(* IEC 61131-3 sources: Lasal/CPU_5344_V01/Class/Lees10Ingangenin, 1 file *)

(* ---- Lees10Ingangenin.st ---- *)
(*!
<Class
	Name               = "Lees10Ingangenin"
	Revision           = "0.0"
	RealtimeTask       = "false"
	CyclicTask         = "false"
	BackgroundTask     = "false"
	Sigmatek           = "false"
	OSInterface        = "false"
	HighPriority       = "false"
	Automatic          = "false"
	UpdateMode         = "Prescan"
	SharedCommandTable = "true"
	Objectsize         = "(284,120)">
	<Channels>
		<Server Name="ClassSVR" Visualized="false" Initialize="false" WriteProtected="true" Retentive="false"/>
		<Client Name="ingang1" Required="false" Internal="false"/>
		<Client Name="ingang10" Required="false" Internal="false"/>
		<Client Name="ingang2" Required="false" Internal="false"/>
		<Client Name="ingang3" Required="false" Internal="false"/>
		<Client Name="ingang4" Required="false" Internal="false"/>
		<Client Name="ingang5" Required="false" Internal="false"/>
		<Client Name="ingang6" Required="false" Internal="false"/>
		<Client Name="ingang7" Required="false" Internal="false"/>
		<Client Name="ingang8" Required="false" Internal="false"/>
		<Client Name="ingang9" Required="false" Internal="false"/>
		<Client Name="Invert" Required="false" Internal="false"/>
	</Channels>
</Class>
*)
Lees10Ingangenin : CLASS
  //Servers:
	ClassSVR 	: SvrChCmd_DINT;
  //Clients:
	ingang1 	: CltCh_DINT;
	ingang2 	: CltCh_DINT;
	ingang3 	: CltCh_DINT;
	ingang4 	: CltCh_DINT;
	ingang5 	: CltCh_DINT;
	ingang6 	: CltCh_DINT;
	ingang7 	: CltCh_DINT;
	ingang8 	: CltCh_DINT;
	ingang9 	: CltCh_DINT;
	ingang10 	: CltCh_DINT;
	Invert 	: CltCh_DINT;
  //Variables:
		gang1 	: DINT;
		gang2 	: DINT;
		gang3 	: DINT;
		gang4 	: DINT;
		gang5 	: DINT;
		gang6 	: DINT;
		gang7 	: DINT;
		gang8 	: DINT;
		gang9 	: DINT;
		gang10 	: DINT;
  //Functions:

	FUNCTION VIRTUAL GLOBAL ClassSVR::Read
		VAR_OUTPUT
			output (EAX) 	: DINT;
		END_VAR;
  //Tables:
	FUNCTION @STD
		VAR_OUTPUT
			ret_code	: CONFSTATES;
		END_VAR;
	FUNCTION GLOBAL TAB @CT_;
END_CLASS;

// JdK 22-7-2019 Lees10IngangenIn, copied from 4090 to 4284
// needs to be translated to English some time

FUNCTION VIRTUAL GLOBAL Lees10Ingangenin::ClassSVR::Read
	VAR_OUTPUT
		output (EAX) 	: DINT;
	END_VAR

  ClassSVR := 0;
  ingang1 := ingang1.Read();
  ingang2 := ingang2.Read();
  ingang3 := ingang3.Read();
  ingang4 := ingang4.Read();
  ingang5 := ingang5.Read();
  ingang6 := ingang6.Read();
  ingang7 := ingang7.Read();
  ingang8 := ingang8.Read();
  ingang9 := ingang9.Read();
  ingang10 := ingang10.Read();
  //alle tweetjes zijn cilinders die niet retour zijn, deze nul maken
  if ingang1 = 2 then ingang1 := 0; end_if;
  if ingang2 = 2 then ingang2 := 0; end_if;
  if ingang3 = 2 then ingang3 := 0; end_if;
  if ingang4 = 2 then ingang4 := 0; end_if;
  if ingang5 = 2 then ingang5 := 0; end_if;
  if ingang6 = 2 then ingang6 := 0; end_if;
  if ingang7 = 2 then ingang7 := 0; end_if;
  if ingang8 = 2 then ingang8 := 0; end_if;
  if ingang9 = 2 then ingang9 := 0; end_if;
  if ingang10 = 2 then ingang10 := 0; end_if;

  Invert := Invert.Read();
  if Invert = 1 then
    gang1 := ingang1=0;
    gang2 := ingang2=0;
    gang3 := ingang3=0;
    gang4 := ingang4=0;
    gang5 := ingang5=0;
    gang6 := ingang6=0;
    gang7 := ingang7=0;
    gang8 := ingang8=0;
    gang9 := ingang9=0;
    gang10 := ingang10=0;
  else
    gang1 := ingang1;
    gang2 := ingang2;
    gang3 := ingang3;
    gang4 := ingang4;
    gang5 := ingang5;
    gang6 := ingang6;
    gang7 := ingang7;
    gang8 := ingang8;
    gang9 := ingang9;
    gang10 := ingang10;
  end_if;
  ClassSVR += gang1 * 1;
  ClassSVR += gang2 * 10;
  ClassSVR += gang3 * 100;
  ClassSVR += gang4 * 1000;
  ClassSVR += gang5 * 10000;
  ClassSVR += gang6 * 100000;
  ClassSVR += gang7 * 1000000;
  ClassSVR += gang8 * 10000000;
  ClassSVR += gang9 * 100000000;
  ClassSVR += gang10 * 1000000000;
	output := ClassSVR;

END_FUNCTION
